TYPE ST_M001_IO_IN :
STRUCT	
	// inputs	
	//bPwrCircBreakerOk	: BOOL;
END_STRUCT
END_TYPE

(* stored: Version 1.1.0.1
   DUT ST_M001_IO_IN: Id {8be6afb1-3284-4976-afe2-961639e6bd4b} *)
